# EPICS substitutions: epics/ioc/sampleIOC/TestIOCApp/Db/user.substitutions
# Example substitutions file

file "db/circle.db" {
    { user = "dphan" }
}

file "db/dbExample1.db" {
    { user = "dphan" }
}

file db/dbExample2.db {
    pattern { user, no, scan }
        { "dphan", 1, "1 second" }
        { "dphan", 2, "2 second" }
        { "dphan", 3, "5 second" }
}
